// TIA Portal V20 export
DATA_BLOCK "db_1"   // DB1
{ S7_Optimized_Access := 'TRUE' }
// stored: MemoryReserve 100
   VAR
      var_1 : Bool;
      var_2 : Int;
      var_3 : Real;
      var_4 : Array[0..9] of Bool;
      var_5 : Bool;
      var_6 : Bool;
      var_7 : Bool;
   END_VAR
BEGIN
END_DATA_BLOCK
